FUNCTION_BLOCK Stage16 (* Template for a Basic Function Block Type *)
  (* Standard: 61499-2 *)
  (* Version 1.0, 2021-06-20, HP *)
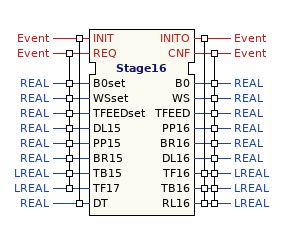
  EVENT_INPUT
    INIT WITH DT; (* Initialization Request *)
    REQ WITH B0set, WSset, TFEEDset, DL15, PP15, BR15, TB15, TF17; (* Normal Execution Request *)
  END_EVENT
  EVENT_OUTPUT
    INITO WITH TB16, RL16, TF16; (* Initialization Confirm *)
    CNF WITH TB16, DL16, TF16, BR16, PP16, TFEED, B0, WS, RL16; (* Execution Confirmation *)
  END_EVENT
  VAR_INPUT
    B0set : REAL;
    WSset : REAL;
    TFEEDset : REAL;
    DL15 : REAL;
    PP15 : REAL;
    BR15 : REAL;
    TB15 : LREAL;
    TF17 : LREAL;
    DT : REAL;
  END_VAR
  VAR_OUTPUT
    B0 : REAL;
    WS : REAL;
    TFEED : REAL;
    PP16 : REAL;
    BR16 : REAL;
    DL16 : REAL;
    TF16 : LREAL;
    TB16 : LREAL;
    RL16 : LREAL;
  END_VAR
  VAR
    AB : REAL; (* internal variabel *)
    UU : REAL;
    TREF : REAL;
    AD : REAL;
    AHC : REAL;
    AHR : REAL;
    AS : REAL;
    REC : REAL;
    WN : REAL;
    WN_1 : REAL;
    XKN : REAL;
    C1 : REAL;
    HS : REAL;
    G : REAL;
    W1 : REAL;
    TFREC : REAL;
    TS : REAL;
    DTS : REAL;
    TF16_last : REAL;
    RL16_last : REAL;
    TB16_last : REAL;
    USS : REAL;
    RHOB : REAL;
    CPB : REAL;
    CPF : REAL;
    FMW : REAL;
    HLV : REAL;
    HV : REAL;
    BPR : REAL;
    FMC : REAL;
    U : REAL;
    A : REAL;
    B : REAL;
    C : REAL;
    D1 : REAL;
    d : REAL;
    a : REAL;
    A1 : REAL;
    A2 : REAL;
    A3 : REAL;
    A4 : REAL;
    A5 : REAL;
    A6 : REAL;
    p : REAL;
    q : REAL;
    TC : REAL;
    PC : REAL;
    DTB16 : REAL;
    DEN16 : REAL;
    DH16 : REAL;
    DP16 : REAL;
    DPDH16 : REAL;
    DT16 : REAL;
    m : REAL;
    n : REAL;
    VR16 : REAL;
    DELTA16 : REAL;
    DELTA38 : REAL;
    DELTA60 : REAL;
    DELTA16_last : REAL;
    DELTA38_last : REAL;
    DELTA60_last : REAL;
  END_VAR
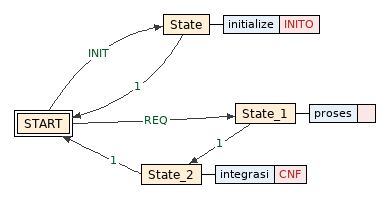
  EC_STATES
    START; (* Initial State *)
    State : initialize -> INITO;
    State_1 : proses;
    State_2 : integrasi -> CNF;
  END_STATES
  EC_TRANSITIONS
    START TO State := INIT;
    State TO START := 1;
    START TO State_1 := REQ;
    State_1 TO State_2 := 1;
    State_2 TO START := 1;
  END_TRANSITIONS
  ALGORITHM initialize IN ST: (* Initialization algorithm *)
TREF :=273.15;
AB :=57.2727;
AHC :=4069.2;
AHR :=2639.7;
AS :=3225.7;
REC :=0.0;
//TF2:=TF2;

//TFEED :=TFEED1+TREF;
 //TS:=TS1+TREF;
WN :=3.0;
XKN :=0.68;
HS:=0.11;
G :=9.81;
W1 :=0.50;

RL16 := 0.609146398558754;
TB16 := 325.755350803451;
TF16 := 322.379704977734;
TF17 := 320.275377684374;



RL16_last :=RL16;
TB16_last :=TB16;
TF16_last :=TF16;
  END_ALGORITHM
  ALGORITHM proses IN ST: (* kalkulasi *)
B0 :=B0set;
WS :=WSset;
TFEED:=TFEEDset;
UU := TFEEDset;
U :=UU;

USS :=49.767;
C1 :=0.625;
RHOB :=1032.4; //maassa jenis brine
CPB :=1.00; //heatcapacity Brine
CPF :=1.00; //heat capacity feed
FMW :=23654.0;
HLV :=563.7959;
HV :=625.1971;
BPR :=2.192;
FMC :=34736.09;
//U :=UU; //feed temp



///  Calculate the physical properties

//A :=3.2437814;
//B :=5.86826*0.001;
//C :=1.1702379*0.00000001;
//D1 :=2.1878462*0.001;
//TC :=647.27;
//PC :=218.167;


A1 :=3.2437814;
A2:=5.86826*0.001;
A3:=1.1702379*0.00000001;
A4 :=2.1878462*0.001;
A5 :=647.27;
A6 :=218.167;

DTB16 :=A5-TB16;
DEN16 :=(A1+A2*DTB16+A3*DTB16*DTB16*DTB16)/(1+A4*DTB16)*DTB16/TB16;
p:=DEN16;
q:=10.0;
PP16 :=A6/(EXPT(q, p));

// calculate the brine flow rates
DP16:=PP15-PP16;
DH16:=RL16-C1*HS;
DPDH16 :=DP16*101000+G*RHOB*DH16;
m:=DPDH16*RHOB;
n:=0.5;
BR16 :=WN*XKN*RL16*(EXPT(m, n));
BR16 :=BR16*60.0/1000.0;

// calculate the vapor flow rates

DT16 :=TB16-BPR/1.8-(TF17+TF16)*0.5;
VR16:=U*AHC*DT16/HLV/1000.0;
DL16 :=DL15+VR16;


//// state equation
DELTA16 :=(BR15-BR16-VR16)*1000.0/RHOB/AB;
DELTA38 :=((BR15*CPB*(TB15-TB16))-VR16*(HV-CPB*(TB16-TREF)))*1000.0/AB/RHOB/CPB/RL16;
DELTA60 :=(B0*CPF*(TF17-TF16)*1000+(U*AHC*DT16))/FMW/CPF;
  END_ALGORITHM
  ALGORITHM integrasi IN ST: (* new algorithm *)
B0 :=B0set;
WS :=WSset;
TFEED:=TFEEDset;
//integrasi
RL16 := (DELTA16 + DELTA16_last)*0.5*DT + RL16_last;
DELTA16_last :=DELTA16 ;
RL16_last :=RL16;

TB16:= (DELTA38 + DELTA38_last)*0.5*DT + TB16_last;
DELTA38_last :=DELTA38 ;
TB16_last:=TB16;

TF16 := (DELTA60 + DELTA60_last)*0.5*DT + TF16_last;
DELTA60_last :=DELTA60 ;
TF16_last :=TF16;
  END_ALGORITHM
END_FUNCTION_BLOCK
